INTERFACE I_TestFrameWorkAdapter

PROPERTY sTestName : REFERENCE TO T_MaxString
GET
END_GET
END_PROPERTY

PROPERTY sTestSuiteName : REFERENCE TO T_MaxString
GET
END_GET
END_PROPERTY

METHOD Verify : HRESULT
VAR_INPUT
	anyArg	: ANY;
END_VAR
END_METHOD

END_INTERFACE

(* stored: Version 1.1.0.1, ProductVersion 3.1.4026.18
   Itf I_TestFrameWorkAdapter: Id {8a43fa44-08f3-4a84-bcbd-9c0d3161876d}
   Property sTestName: Id {9630ba0e-b1f6-4c82-bd5f-2832aef2b56b}
   Get Get: Id {73e38f85-ca52-4b13-9e22-bb66d3c01cf6}
   Property sTestSuiteName: Id {8bf4ff20-5ce5-4689-ac1a-2bf0b58b9021}
   Get Get: Id {1106f76c-b8d2-48d6-a255-5df9e4d49fbb}
   Method Verify: Id {31977d99-b7f0-467b-8866-c72c42cc6436} *)
